// TIA Portal V17 export
// export: Created 2024-08-07T21:44:14.2356687Z, ExportSetting WithDefaults, DisplayName Totally Integrated Automation Portal, DisplayVersion V17 Update 7, DisplayName TIA Portal Openness, DisplayVersion V17 Update 7, DisplayName TIA Portal Version Control Interface, DisplayVersion V17, DisplayName SINAMICS Startdrive Advanced, DisplayVersion V17 SP2, DisplayName SINAMICS Startdrive G110M, G120, G120C, G120D, G120P, G115D, DisplayVersion V17 SP2, DisplayName SINAMICS Startdrive G130, G150, S120, S150, SINAMICS MV, S210, DisplayVersion V17 SP2, DisplayName STEP 7 Professional, DisplayVersion V17 Update 7, DisplayName STEP 7 Safety, DisplayVersion V17 Update 6, DisplayName WinCC Advanced / Unified PC, DisplayVersion V17 Update 7
TYPE "UDT_DateTimeAndShiftsSettings"
// stored: IsFailsafeCompliant false
   STRUCT
      DateAndTime : DTL := DTL#2019-01-17-00:00:00;   // Date and time to set
      Shift1Enabled : Bool := TRUE;   // Shift 1 enabled: 0= No,
      Shift1StartTime : Time_Of_Day := TOD#6:0:0.000;   // Shift 1 start time
      Shift1EndTime : Time_Of_Day := TOD#14:0:0.000;   // Shift 1 end time
      Shift2Enabled : Bool := TRUE;   // Shift 2 enabled: 0= No
      Shift2StartTime : Time_Of_Day := TOD#14:0:0.000;   // Shift 2 start time
      Shift2EndTime : Time_Of_Day := TOD#22:0:0.000;   // Shift 2 end time
      Shift3Enabled : Bool := TRUE;   // Shift 3 enabled: 0= No
      Shift3StartTime : Time_Of_Day := TOD#22:0:0.000;   // Shift 3 start time
      Shift3EndTime : Time_Of_Day := TOD#6:0:0.000;   // Shift 3 end time
   END_STRUCT;
END_TYPE
